{attribute 'qualified_only'}
VAR_GLOBAL
	

	Setting: ARRAY[0..constcsv.MAX_SETTING_LENGTH] OF typeSettings;
	
	varSelectedColumn:INT;
	varSelectedRow:INT;
	
	varSelectedColumnValid:BOOL;
	varSelectedRowValid:BOOL;
	
	btnRead:BOOL;
	btnWrite:BOOL;
	
	numElementsOfSettings:INT;
	
	numSelectedSetting:INT;
	numSelectedSettingNew:INT;
	btnMoveValue:BOOL;
	
	
	
END_VAR

(* stored: Version 1.1.0.1, ProductVersion 3.1.4024.11
   GVL MachineSettings: Id {e5f65bc7-f264-06b6-333b-91c362883b10} *)
